FUNCTION_BLOCK FB_CoolingControl

VAR
	_bInit			: BOOL;
	
	_refHmi			: REFERENCE TO ST_CoolingControlHmi;
	_iMotor			: I_Motor;
	_iRoomTemp		: I_RoomTemp;
	
	eCoolingState	: E_CoolingControlState;
	
	_fbBasicPID		: FB_BasicPID;
	_nPidOut		: LREAL;
	_nPidOutAbs		: LREAL;
END_VAR

// rajapinnan kautta valvotaan huoneen läpmötilaa. keksitään PID yms säädin, joka nostaa tamun tehoja 
// kun lämpötila nousee...

IF _iMotor.bAuto AND _refHmi.bAuto THEN
	eCoolingState := E_CoolingControlState.Auto;
	
ELSIF NOT _iMotor.bAuto THEN
	eCoolingState := E_CoolingControlState.Manual;
	
	
END_IF

StateMachine();

//FB_Init is always available implicitly and it is used primarily for initialization.
//The return value is not evaluated. For a specific influence, you can also declare the
//methods explicitly and provide additional code there with the standard initialization
//code. You can evaluate the return value.
METHOD FB_Init: BOOL
VAR_INPUT
    bInitRetains: BOOL; // TRUE: the retain variables are initialized (reset warm / reset cold)
    bInCopyCode: BOOL;  // TRUE: the instance will be copied to the copy code afterward (online change)   
END_VAR
_bInit := TRUE;
END_METHOD

METHOD Init : BOOL
VAR_INPUT
	
	refHmi			: REFERENCE TO ST_CoolingControlHmi;
	sName			: STRING;
	iMotor			: I_Motor;
	iRoomTemp		: I_RoomTemp;
END_VAR
IF _bInit THEN
	
	_refHmi			REF= refHmi;
	_refHmi.sName	:= sName;
	_iMotor			:= iMotor;
	_iRoomTemp		:= iRoomTemp;





	_bInit := FALSE;
		
END_IF
END_METHOD

METHOD PRIVATE MotorControl
VAR_INPUT
END_VAR
END_METHOD

METHOD PRIVATE StateMachine : BOOL
VAR_INPUT
END_VAR
CASE eCoolingState OF
	
	E_CoolingControlState.Auto:
		IF _iRoomTemp.nRoomTemp > _refHmi.paramRoomTempSet THEN
			
			_fbBasicPID(	fSetpointValue:= REAL_TO_LREAL(_refHmi.paramRoomTempSet), 
							fActualValue:= REAL_TO_LREAL(_iRoomTemp.nRoomTemp), 
							bReset:= 0, 
							fCtrlCycleTime:= 0.01, 
							fKp:= _refHmi.param_P, 
							fTn:= _refHmi.param_I, 
							fTv:= _refHmi.Param_D, 
							fTd:= 0, 
							fCtrlOutput=> _nPidOut, 
							nErrorStatus=> );
							
							_nPidOutAbs := ABS(_nPidOut);
							_iMotor.nSpeed := LREAL_TO_INT( MAX(0.0, MIN(100.0, _nPidOutAbs)));
							
		END_IF
		
		IF _nPidOutAbs > 5 THEN
		_iMotor.bEnable := TRUE;
		END_IF
		
		
	E_CoolingControlState.Manual:
	;
	
	E_CoolingControlState.Stop:
	;
	
	E_CoolingControlState.Error:
	;
	
END_CASE
END_METHOD

END_FUNCTION_BLOCK

(* stored: Version 1.1.0.1
   POU FB_CoolingControl: Id {c09f89a4-7fd2-41a6-a90f-53be9d89a7cd}, SpecialFunc None
   Method FB_Init: Id {fcfc5886-4c00-430c-bcfe-6efe2b92512a}
   Method Init: Id {41d1ef6e-1d92-4a89-a068-5cd5a1e489d5}
   Method MotorControl: Id {fca439e2-536d-4a5e-b82f-23ba2cccf372}
   Method StateMachine: Id {fc3a95a4-aa4c-4d2d-b42b-fbab5f8880e3} *)
